FUNCTION_BLOCK TcoContext_Waveform EXTENDS TcoContext
VAR
	_TcoObject_Waveform		:	TcoObject_Waveform(THIS^);
END_VAR

METHOD PROTECTED  Main
_TcoObject_Waveform();
END_METHOD

END_FUNCTION_BLOCK

(* stored: Version 1.1.0.1, ProductVersion 3.1.4024.5
   POU TcoContext_Waveform: Id {75ef8a24-aecd-4e0a-addd-347a92f690b1}, SpecialFunc None
   Method Main: Id {247c75f9-f2be-4116-80b6-fa8029df4445} *)
